INTERFACE I_AsyncManagerConfig

METHOD PUBLIC TryGetSessionIdFromResponse : BOOL
VAR_INPUT
	Response : I_ServerResponse;
	Destination : ANY;
END_VAR
END_METHOD

END_INTERFACE

(* stored: Version 1.1.0.1, ProductVersion 3.1.4024.12
   Itf I_AsyncManagerConfig: Id {4a4f0798-ed83-499b-b5a8-20a54d5c473a}
   Method TryGetSessionIdFromResponse: Id {86bdc0c7-ab84-4ab2-b087-c91b835ef3a4} *)
